TYPE T_FileAccessMode : DWORD; END_TYPE

(* stored: Version 1.1.0.1, ProductVersion 3.1.4024.14
   DUT T_FileAccessMode: Id {edd73d5f-33f1-0bc0-2cb0-a64530c8b817} *)
